TYPE ST_MKS_925 EXTENDS ST_VacuumGauge :
STRUCT
END_STRUCT
END_TYPE

(* stored: Version 1.1.0.1, ProductVersion 3.1.4019.2
   DUT ST_MKS_925: Id {432a3417-2042-4dcd-9dc9-c4ee7d4a0ebb} *)
